INTERFACE I_InterfaceDatatype EXTENDS I_Datatype

PROPERTY PUBLIC Identifier : T_MAXSTRING
GET
END_GET
END_PROPERTY

END_INTERFACE

(* stored: Version 1.1.0.1, ProductVersion 3.1.4024.12
   Itf I_InterfaceDatatype: Id {9ab490f0-4162-461c-a7e3-468cf80da484}
   Property Identifier: Id {c4d1e14d-966f-49cb-9ac2-26d0d290aa63}
   Get Get: Id {004e6a33-bcc0-44c3-8352-5d5caff9b5ea} *)
